{attribute addProperty BoxType "EPP1332-0001-0016"}
{attribute addProperty Id "A_0022_EPP1332_0001_0017A_0022_EPP1332_0001_0017_4E5F00D52662332.75"}
{attribute addProperty CRC "209047392"}
{attribute addProperty SizeInBites "2662"}
{attribute addProperty SizeInBytes "332.75"}
TYPE A_0021_EPP1332_0001_0016_0C75CF60 EXTENDS EPP1332_179A0949 :
STRUCT
	{attribute addProperty Name "A_0022_EPP1332_0001_0017"}
	A_0022_EPP1332_0001_0017 : A_0022_EPP1332_0001_0017_4E5F00D5;
END_STRUCT
END_TYPE

(* stored: Version 1.2.0.0, ProductVersion 3.1.4024.9
   DUT A_0021_EPP1332_0001_0016_0C75CF60: Id {e48a9a4a-395a-488a-909a-e31459add206} *)
